FUNCTION_BLOCK FB_MBusReadInputRegs EXTENDS FB_MBusFunc
VAR_INPUT
	nNumOfInputRegs		: WORD;
	nStartAddr			: WORD;
END_VAR
VAR_OUTPUT
	nInputReg0			: INT;
	nInputReg1			: INT;
	nInputReg2			: INT;
	nInputReg3			: INT;
	nInputReg4			: INT;
	nInputReg5			: INT;
	nInputReg6			: INT;
	nInputReg7			: INT;
END_VAR
VAR
	fbMBReadInputRegs	: FB_MBReadInputRegs;
	aReadBuffer			: ARRAY[0..7] OF INT;
END_VAR

SUPER^();

METHOD PROTECTED  CallMBFunc
VAR_INPUT
END_VAR
fbMBReadInputRegs(
	bExecute := FALSE,
	bBusy=> stMBusStatus.bBusy, 
	bError=> stMBusStatus.bError, 
	nErrId=> stMBusStatus.nErrId
);
END_METHOD

METHOD PROTECTED  ClearFBOutput
VAR_INPUT
END_VAR
nInputReg0 := 0;
nInputReg1 := 0;
nInputReg2 := 0;
nInputReg3 := 0;
nInputReg4 := 0;
nInputReg5 := 0;
nInputReg6 := 0;
nInputReg7 := 0;
END_METHOD

METHOD PROTECTED  ReadFBInput
VAR_INPUT
END_VAR
// Do nothing
END_METHOD

METHOD PROTECTED  TriggerMBFunc
VAR_INPUT
END_VAR
fbMBReadInputRegs(
	sIPAddr:= stMBUSConnection.sIPAddr, 
	nTCPPort:= stMBUSConnection.nTCPPort, 
	nUnitID:= stMBUSConnection.nUnitID, 
	nQuantity:= nNumOfInputRegs, 
	nMBAddr:= nStartAddr, 
	cbLength:= SIZEOF(aReadBuffer), 
	pDestAddr:= ADR(aReadBuffer), 
	bExecute:= TRUE, 
	tTimeout:= stMBUSConnection.tTimeout, 
	bBusy=> stMBusStatus.bBusy, 
	bError=> stMBusStatus.bError, 
	nErrId=> stMBusStatus.nErrId, 
	cbRead=> );
END_METHOD

METHOD PROTECTED  WriteFBOutput
VAR_INPUT
END_VAR
nInputReg0 := aReadBuffer[0];
nInputReg1 := aReadBuffer[1];
nInputReg2 := aReadBuffer[2];
nInputReg3 := aReadBuffer[3];
nInputReg4 := aReadBuffer[4];
nInputReg5 := aReadBuffer[5];
nInputReg6 := aReadBuffer[6];
nInputReg7 := aReadBuffer[7];
END_METHOD

END_FUNCTION_BLOCK

(* stored: Version 1.1.0.1, ProductVersion 3.1.4024.15
   POU FB_MBusReadInputRegs: Id {17e9d00e-d975-48c3-884f-07cc9bbf41b1}, SpecialFunc None
   Method CallMBFunc: Id {5bc94b6c-7b40-4655-8c73-0ac7d72ad3c6}
   Method ClearFBOutput: Id {1ff09b27-c820-4f70-9620-612b7aa4b4df}
   Method ReadFBInput: Id {71417c77-e6f6-4959-b077-0c4b6cb097c9}
   Method TriggerMBFunc: Id {3f48e448-409d-4cbf-ac29-5b6d6a73026a}
   Method WriteFBOutput: Id {3dc3f4d6-4a6f-4494-bd2d-3778babc5004} *)
